VAR_GLOBAL
	//Deck 1
	//Drive inputs
	ATV_State_D4							AT	%I*		: WORD; //Drive state
	ATV_TPDO_Input1_Status_Word_D4			AT	%I*		: WORD;	//Status Word From Drive
	iVelocityRaw_D4							AT	%I*		: INT;	//Velocity From Drive - Address 8604 - Units 1 RPM
	iTorqueRaw_D4							AT	%I*		: INT;	//Torque From Drive - Address 3205 - Units 0.1%
	uiCurrentRaw_D4							AT	%I*		: UINT;	//Current From Drive - Address 3204 - Units 0.1A
	uiVoltageRaw_D4							AT	%I*		: UINT;	//Voltage From Drive - Address 3208 - Units 1V
	uiFaultCode_D4							AT	%I*		: UINT;	//Fault Codes
	//End drive inputs	
	
	//Drive outputs
	ATV_RPDO_Output1_Control_Word_D4		AT	%Q*		: WORD;	//Control Word To Drive
	ATV_RPDO_Output2_Target_Velocity_D4		AT	%Q*		: WORD; //Velocity To Drive in RPM - Max Value 32767
	//End drive outputs

	//Inputs Status Word Bit Level
	xReady_To_Switch_on_D4 								: BOOL;//Bit 0
	xSwitched_ON_D4										: BOOL;//Bit 1
	xOperationEnabled_D4 								: BOOL;//Bit 2
	xFault_D4 											: BOOL;//Bit 3
	xVoltageEnabled_D4									: BOOL;//Bit 4
	xQuickStop_D4										: BOOL;//Bit 5
	xSwitchOnDisabled_D4 								: BOOL;//Bit 6
	xWarning_D4											: BOOL;//Bit 7
	xTargetReached_D4									: BOOL;//Bit 10
	xInternalLimitActive_D4								: BOOL;//Bit 11
	xDirectionofRotation_D4								: BOOL;//Bit 15	
	stFault_D4											: STRING;
	rTorqueValue_D4										: REAL;
	rCurrentValue_D4									: REAL;
	lrSpeed_D4											: LREAL;
	xEnable_D4											: BOOL; //Enable Drive Trigger
	xStart_D4											: BOOL;	//Start Trigger
	xStop_D4 											: BOOL;	//Stop Trigger
	iDirection_D4										: INT;	//Direction	Trigger
	xForward_D4											: BOOL; //Forward Trigger
	xReverse_D4											: BOOL;	//Reverse Trigger
	xReset_D4											: BOOL;	//Reset Trigger
	xInputStatus_HMI_D4									: ARRAY [0..9] OF BOOL;	//VFD Status Bits
	//End inputs Status Word Bit Level
	//End Deck 1
END_VAR

(* stored: Version 1.1.0.1, ProductVersion 3.1.4024.3
   GVL Deck4: Id {63d50a48-f32b-4c92-af26-5d4db90d826f} *)
